Staubli VAL3: rightPos.pgx

public program rightPos(string x_sItem (dimensions=1), num x_nLength (dimensions=1), string& x_sResult[] (dimensions=1))
  local num i
  local num l_nLength
  local string l_sItem
begin
  //
  l_sItem=x_sItem
  // divide the string...
  if len(l_sItem)!=getDisplayLen(l_sItem) and x_nLength<=getDisplayLen(l_sItem) and x_nLength>0
    for i=len(x_sItem)-1 to 0 step -1
      l_nLength=l_nLength+getDisplayLen(right(l_sItem,1))
      l_sItem=left(l_sItem,len(l_sItem)-1)
      if l_nLength==x_nLength
        x_sResult=right(x_sItem,len(x_sItem)-i)
        return
      else
        if l_nLength>x_nLength
          x_sResult=right(x_sItem,len(x_sItem)-i-1)
          return
        endIf
      endIf
    endFor
  endIf
  //else
  x_sResult=right(x_sItem,max(x_nLength,0))
  //endIf
end
